// TIA Portal V17 export
// export: Created 2024-08-29T18:23:43.5796752Z, ExportSetting WithDefaults, DisplayName Totally Integrated Automation Portal, DisplayVersion V17 Update 7, DisplayName TIA Portal Openness, DisplayVersion V17 Update 7, DisplayName TIA Portal Version Control Interface, DisplayVersion V17, DisplayName SINAMICS Startdrive Advanced, DisplayVersion V17 SP2, DisplayName SINAMICS Startdrive G110M, G120, G120C, G120D, G120P, G115D, DisplayVersion V17 SP2, DisplayName SINAMICS Startdrive G130, G150, S120, S150, SINAMICS MV, S210, DisplayVersion V17 SP2, DisplayName STEP 7 Professional, DisplayVersion V17 Update 7, DisplayName STEP 7 Safety, DisplayVersion V17 Update 6, DisplayName WinCC Advanced / Unified PC, DisplayVersion V17 Update 7
DATA_BLOCK "eks"   // DB305
{ S7_Optimized_Access := 'FALSE' }
VERSION : 0.1
// stored: AutoNumber false, DBAccessibleFromOPCUA true, DBAccessibleFromWebserver true, IsOnlyStoredInLoadMemory false, IsWriteProtectedInAS false
   VAR RETAIN
      status : Struct
         operator : Bool := TRUE;
         gapLeader : Bool := TRUE;
         maintenance : Bool := TRUE;
         administrator : Bool := TRUE;
         spare4 : Bool := FALSE;
         spare5 : Bool := FALSE;
         spare6 : Bool := FALSE;
         spare7 : Bool := FALSE;
         addModeEnabled : Bool := TRUE;
         addMode : Bool := FALSE;
         reset : Bool := FALSE;
         nbMaxAchieved : Bool := FALSE;
         fpStoreKeyIn : Bool := FALSE;
         spare15 : Bool := FALSE;
         spare16 : Bool := FALSE;
         spare17 : Bool := FALSE;
      END_STRUCT;
      hmi : Struct
         operatorKey : Bool := FALSE;
         addMode : Bool := FALSE;
         endAddMode : Bool := FALSE;
         writeKeyNewLevel : Bool := FALSE;
         writeKewKeyID : Bool := FALSE;
         updateNbAdmin : Bool := FALSE;
         spare6 : Bool := FALSE;
         spare7 : Bool := FALSE;
         spare10 : Bool := FALSE;
         spare11 : Bool := FALSE;
         spare12 : Bool := FALSE;
         spare13 : Bool := FALSE;
         spare14 : Bool := FALSE;
         spare15 : Bool := FALSE;
         spare16 : Bool := FALSE;
         spare17 : Bool := FALSE;
      END_STRUCT;
      timeout : Struct
         resetSet : Int := 9999;
         resetStatus : Int := 9100;
      END_STRUCT;
      pageIndex : Int := 1;   // Index of the page of HMI
      saveLine : Int := 0;   // Line to save key
      removeLine : Int := 0;   // Line to remove key
      actualLevel : Int := 5;   // Actual level of key
      nbAdmin : Int := 30740;   // Number of admin counted
      tCycle : Int := 0;   // Index for function Cycle (look for key)
      nbMaxAdmin : Int := 5;   // Number of administrator max
      savedPageNumber : Word := 16#0001;
      sparesBlock1 : Array[22..47] of Byte;   // Reserve
      insertedKey { S7_SetPoint := 'True'} : "udt_EKS_KEY";   // Information of Key Inserted
      hmiPage { S7_SetPoint := 'True'} : Array[1..10] of "udt_EKS_KEY";   // Information displayed on HMI
      spareBlock2 : Array[270..299] of Byte;   // Reserve
      keys { S7_SetPoint := 'True'} : Array[1..130] of "udt_EKS_KEY";
      deleteKeys : "udt_EKS_KEY";
   END_VAR
BEGIN
   sparesBlock1[22..47] := 16#00;
   insertedKey.ID1 := 16#6B8F_0010;
   insertedKey.ID2 := 16#3200_0000;
   insertedKey.EMPLOYEE_ID := 16#0000_0000;
   insertedKey.LEVEL := 5;
   insertedKey.COMMENTS := WSTRING#'ADMIN';
   insertedKey._res_1 := 0;
   hmiPage[1].ID1 := 16#27A0_0010;
   hmiPage[2].ID1 := 16#8DDD_0010;
   hmiPage[3].ID1 := 16#9750_0010;
   hmiPage[4].ID1 := 16#4D33_0010;
   hmiPage[5].ID1 := 16#7650_0010;
   hmiPage[6].ID1 := 16#6B8F_0010;
   hmiPage[7].ID1 := 16#3A6D_0010;
   hmiPage[8..10].ID1 := 16#0000_0000;
   hmiPage[1..7].ID2 := 16#3200_0000;
   hmiPage[8..10].ID2 := 16#0000_0000;
   hmiPage[1].EMPLOYEE_ID := 16#0001_0000;
   hmiPage[2].EMPLOYEE_ID := 16#0000_0001;
   hmiPage[3].EMPLOYEE_ID := 16#0000_0002;
   hmiPage[4..5].EMPLOYEE_ID := 16#0000_0000;
   hmiPage[6].EMPLOYEE_ID := 16#0000_0200;
   hmiPage[7].EMPLOYEE_ID := 16#0000_0100;
   hmiPage[8..10].EMPLOYEE_ID := 16#0000_0000;
   hmiPage[1].LEVEL := 5;
   hmiPage[2].LEVEL := 2;
   hmiPage[3].LEVEL := 3;
   hmiPage[4].LEVEL := 5;
   hmiPage[5].LEVEL := 3;
   hmiPage[6].LEVEL := 5;
   hmiPage[7].LEVEL := 3;
   hmiPage[8..10].LEVEL := 0;
   hmiPage[1].COMMENTS := WSTRING#'CESAR';
   hmiPage[2].COMMENTS := WSTRING#'GAP';
   hmiPage[3].COMMENTS := WSTRING#'MANT';
   hmiPage[4..5].COMMENTS := WSTRING#'CESAR';
   hmiPage[6].COMMENTS := WSTRING#'ADMIN';
   hmiPage[7].COMMENTS := WSTRING#'MANT';
   hmiPage[8..10].COMMENTS := WSTRING#'';
   hmiPage[1..10]._res_1 := 0;
   spareBlock2[270..299] := 16#00;
   keys[1].ID1 := 16#27A0_0010;
   keys[2].ID1 := 16#8DDD_0010;
   keys[3].ID1 := 16#9750_0010;
   keys[4].ID1 := 16#4D33_0010;
   keys[5].ID1 := 16#7650_0010;
   keys[6].ID1 := 16#6B8F_0010;
   keys[7].ID1 := 16#3A6D_0010;
   keys[8..109].ID1 := 16#0000_0000;
   keys[110].ID1 := 16#DB52_0010;
   keys[111..130].ID1 := 16#0000_0000;
   keys[1..7].ID2 := 16#3200_0000;
   keys[8..109].ID2 := 16#0000_0000;
   keys[110].ID2 := 16#3200_0000;
   keys[111..130].ID2 := 16#0000_0000;
   keys[1].EMPLOYEE_ID := 16#0001_0000;
   keys[2].EMPLOYEE_ID := 16#0000_0001;
   keys[3].EMPLOYEE_ID := 16#0000_0002;
   keys[4..5].EMPLOYEE_ID := 16#0000_0000;
   keys[6].EMPLOYEE_ID := 16#0000_0200;
   keys[7].EMPLOYEE_ID := 16#0000_0100;
   keys[8..130].EMPLOYEE_ID := 16#0000_0000;
   keys[1].LEVEL := 5;
   keys[2].LEVEL := 2;
   keys[3].LEVEL := 3;
   keys[4].LEVEL := 5;
   keys[5].LEVEL := 3;
   keys[6].LEVEL := 5;
   keys[7].LEVEL := 3;
   keys[8..109].LEVEL := 0;
   keys[110].LEVEL := 5;
   keys[111..130].LEVEL := 0;
   keys[1].COMMENTS := WSTRING#'CESAR';
   keys[2].COMMENTS := WSTRING#'GAP';
   keys[3].COMMENTS := WSTRING#'MANT';
   keys[4..5].COMMENTS := WSTRING#'CESAR';
   keys[6].COMMENTS := WSTRING#'ADMIN';
   keys[7].COMMENTS := WSTRING#'MANT';
   keys[8..109].COMMENTS := WSTRING#'';
   keys[110].COMMENTS := WSTRING#'Robins';
   keys[111..130].COMMENTS := WSTRING#'';
   keys[1..130]._res_1 := 0;
   deleteKeys.ID1 := 16#0000_0000;
   deleteKeys.ID2 := 16#0000_0000;
   deleteKeys.EMPLOYEE_ID := 16#0000_0000;
   deleteKeys.LEVEL := 0;
   deleteKeys.COMMENTS := WSTRING#'';
   deleteKeys._res_1 := 0;
END_DATA_BLOCK
